// TIA Portal V16 export
// export: Created 2021-11-12T13:32:36.0735124Z, ExportSetting WithDefaults, DisplayName Totally Integrated Automation Portal, DisplayVersion V16 Update 3, DisplayName TIA Portal Version Control Interface, DisplayVersion V16 Update 2, DisplayName TIA Portal Openness, DisplayVersion V16 Update 3, DisplayName SINAMICS Startdrive Advanced, DisplayVersion V16 Update 5, DisplayName SINAMICS Startdrive G130, G150, S120, S150, SINAMICS MV, S210, DisplayVersion V16 Update 5, DisplayName SINAMICS Startdrive G110M, G120, G120C, G120D, G120P, G115D, DisplayVersion V16 Update 5, DisplayName STEP 7 Professional, DisplayVersion V16 Update 3, DisplayName STEP 7 Safety, DisplayVersion V16, DisplayName WinCC UA Professional, DisplayVersion V16 Update 3
DATA_BLOCK "STATUS_210"   // DB2103
{ S7_Optimized_Access := 'TRUE' }
VERSION : 0.1
// stored: AutoNumber false, DBAccessibleFromOPCUA true, IsOnlyStoredInLoadMemory false, IsRetainMemResEnabled false, IsWriteProtectedInAS false, MemoryReserve 100
   VAR
      xxxxx___BinarySensors___xxxxx : Byte;
      xxxxx___BinaryOthers___xxxxx : Byte;
      "UF01-SF02_14" : Bool;   // Dopravník Remote
      "UF01-SF02_24" : Bool;   // Dopravník Automat
      "UF01-SF03_14" : Bool;   // Dopravník Manuál Vzad
      "UF01-SF03_24" : Bool;   // Dopravník Manuál Vpřed
      "UF01-SF04_14" : Bool;   // Dopravník Start automat
      "UF01-SF05_12" : Bool;   // Dopravník Stop
      "UF01-SF07_14" : Bool;   // Bedna Žádost o výměnu
      "UF01-SF08_14" : Bool;   // Bedna Vyměněna
      "UC12-FC01_14" : Bool;   // 400V Dopravník ++210 (L1) OK
      xxxxx___AnalogueSensors___xxxxx : Byte;
      xxxxx___Drives___xxxxx : Byte;
      GL01_MA01 : Struct   // Blank conveyour (L1) - motor / Vyvážecí dopravník přířezů (L1) - motor
         Main { S7_SetPoint := 'True'} : "UDT_Status_main";
         Specific { S7_SetPoint := 'True'} : "UDT_Drive1_Status_specific";
         Error { S7_SetPoint := 'True'} : "UDT_Error01";
      END_STRUCT;
      UC12_TA01 : Struct   // Blank conveyour (L1) - G120 / Vyvážecí dopravník přířezů (L1) - měnič G120
         Main { S7_SetPoint := 'True'} : "UDT_Status_main";
         Specific { S7_SetPoint := 'True'} : "UDT_SINAMICS_G120_Status_specific";
         Error { S7_SetPoint := 'True'} : "UDT_Error02";
      END_STRUCT;
      xxxxx___Others___xxxxx : Byte;
      CL01 : Struct   // Box for blanks / Bedna na přířezy
         Main : "UDT_Status_main";
         Specific : "UDT_PartCounter_Status";
         Error : "UDT_Error01";
      END_STRUCT;
      xxxxx___SensorAlarms___xxxxx : Byte;
      xxxxx___ProcessAlarms___xxxxx : Byte;
      CL01_Alarm : Struct   // CL01 - box full / CL01 - bedna plná.
         Main : "UDT_Status_main";
         Specific : "UDT_DI_Mon_Status_specific";
         Error : "UDT_Error01";
      END_STRUCT;
      CL01_Warn : Struct   // CL01 - box full / CL01 - bedna plná.
         Main : "UDT_Status_main";
         Specific { S7_SetPoint := 'True'} : "UDT_DI_Mon_Status_specific";
         Error { S7_SetPoint := 'True'} : "UDT_Error01";
      END_STRUCT;
      xxxxx__SafetyAlarms__xxxxx : Byte;
      ES : Struct   // E-stop
         Main { S7_SetPoint := 'True'} : "UDT_Status_main";
         Specific { S7_SetPoint := 'True'} : "UDT_DI_Mon_Status_specific";
         Error { S7_SetPoint := 'True'} : "UDT_Error01";
      END_STRUCT;
   END_VAR
BEGIN
END_DATA_BLOCK
